{attribute 'qualified_only'}
VAR_GLOBAL
END_VAR

(* stored: Version 1.1.0.1, ProductVersion 3.1.4022.7
   GVL GVL_03_Delay_Common: Id {18ad61d9-eafe-43dd-bc51-cb5a08ca7d1f} *)
